Fanuc KAREL source: kc00050.KL

-- PROVISIONAL review KL for V940-1; original PC SHA256 25d473540b7f4687345e76c3d10dd2b1a4b23be3f64153bdb2000160d40ff527
-- Incomplete behavior may be omitted. Consult companion uncertainty JSON. Do not deploy.
PROGRAM KC00050
%NOLOCKGROUP
BEGIN
  -- V9_ZERO_TABLE_METADATA_HINT layout=0002_ascii; no indexed target words; source/name/runtime held
  -- UNRESOLVED_PC offsets 5-35; opcodes 27,22,22,1C,22,27,9D,31
  -- UNRESOLVED_PC offsets 40-44; opcodes 7F
END KC00050
